(* IEC 61131-3 sources: inproshop/test8_exported/1.Function/FB/Robot(机械手)/Kuka-六轴, 4 files *)

(* ---- Str_Kuka6.st ---- *)
TYPE Str_Kuka6 :
STRUCT
	Cmd:Str_Kuka6Cmd;//控制
	Status:Str_Kuka6Status;//状态
END_STRUCT
END_TYPE

(* ---- Str_Kuka6Cmd.st ---- *)
TYPE Str_Kuka6Cmd :
STRUCT
	AppID0			:BOOL;//Main程序编号
	AppID1			:BOOL;//Main程序编号
	AppID2			:BOOL;//Main程序编号
	AppID3			:BOOL;//Main程序编号
	AppID4			:BOOL;//Main程序编号
	AppID5			:BOOL;//Main程序编号
	AppID6			:BOOL;//Main程序编号
	AppID7			:BOOL;//Main程序编号
	PGNO_VALID		:BOOL;//程序号有效
	EXT_START		:BOOL;//启动
	MOVE_ENABLE		:BOOL;//运行开通-激活运动使能
	CONF_MESS		:BOOL;//错误确认
	DRIVES_OFF		:BOOL;//驱动器关闭
	DRIVES_ON		:BOOL;//驱动装置接通
	EXT_Stop		:BOOL;//程序复位
	MachineIntial	:BOOL;//设备初始化
	MachineAutoRun	:BOOL;//设备自动中
	MachineStepRun	:BOOL;//单步信号
	SpaceBoo19		:BOOL;//预备位
	SpaceBoo20		:BOOL;//预备位
	SpaceBoo21		:BOOL;//预备位
	SpaceBoo22		:BOOL;//预备位
	SpaceBoo23		:BOOL;//预备位
	SpaceBoo24		:BOOL;//预备位
	SpaceBoo25		:BOOL;//预备位
	SpaceBoo26		:BOOL;//预备位
	SpaceBoo27		:BOOL;//预备位
	SpaceBoo28		:BOOL;//预备位
	SpaceBoo29		:BOOL;//预备位
	SpaceBoo30		:BOOL;//预备位
	SpaceBoo31		:BOOL;//预备位
	SpaceBoo32		:BOOL;//预备位
	InterFace_B		:ARRAY[33..64] OF BOOL;//交互信号
	Speed				:INT;//	运行速度(第9-10个字节)
	ProductType			:INT;//配方型号(第11-12个字节)
	StepNum				:INT;//步序号(第13-14个字节)
	InterFace_Register4	:INT;//交换数据字(第15-16个字节)
	InterFace_Register5	:INT;//交换数据字(第17-18个字节)
	InterFace_Register6	:INT;//交换数据字(第19-20个字节)
	InterFace_Register7	:INT;//交换数据字(第21-22个字节)
	InterFace_Register8	:INT;//交换数据字(第23-24个字节)
	InterFace_Register9	:INT;//交换数据字(第25-26个字节)
	InterFace_Register10	:REAL;//交换数据字(第27-30个字节)
	InterFace_Register11	:REAL;//交换数据字(第31-34个字节)
	InterFace_Register12	:REAL;//交换数据字
	InterFace_Register13	:REAL;//交换数据字
	InterFace_Register14	:REAL;//交换数据字
	InterFace_Register15	:REAL;//交换数据字
	InterFace_Register16	:REAL;//交换数据字

END_STRUCT
END_TYPE

(* ---- Str_Kuka6Status.st ---- *)
TYPE Str_Kuka6Status :
STRUCT
	AppID0			:BOOL;//返回程序编号
	AppID1			:BOOL;//返回程序编号
	AppID2			:BOOL;//返回程序编号
	AppID3			:BOOL;//返回程序编号
	AppID4			:BOOL;//返回程序编号
	AppID5			:BOOL;//返回程序编号
	AppID6			:BOOL;//返回程序编号
	AppID7			:BOOL;//返回程序编号
	ALARM_STOP:		BOOL;//	急停
	USER_SAF:		BOOL;//	安全门
	Ready:			BOOL;//	驱动器处于待机运行状态
	STOPMESS:		BOOL;//	集合故障
	PRO_ACT:		BOOL;//	程序激活
	PGNO_REQ:		BOOL;//	程序号请求
	APPL_RUN:		BOOL;//	运行中
	EXT:			BOOL;//外部自动运行
	Intialed:		BOOL;//	机械手初始化完成
	SpaceBoo18		:BOOL;//预备位
	SpaceBoo19		:BOOL;//预备位
	SpaceBoo20		:BOOL;//预备位
	SpaceBoo21		:BOOL;//预备位
	SpaceBoo22		:BOOL;//预备位
	SpaceBoo23		:BOOL;//预备位
	SpaceBoo24		:BOOL;//预备位
	SpaceBoo25		:BOOL;//预备位
	SpaceBoo26		:BOOL;//预备位
	SpaceBoo27		:BOOL;//预备位
	SpaceBoo28		:BOOL;//预备位
	SpaceBoo29		:BOOL;//预备位
	SpaceBoo30		:BOOL;//预备位
	SpaceBoo31		:BOOL;//预备位
	SpaceBoo32		:BOOL;//预备位
	InterFace_B:ARRAY[33..64] OF BOOL;//交互信号
	ErrorCode:			WORD;//	错误代码（9-10）
	ProductType			:INT;//配方型号(第11-12个字节)
	StepNum				:INT;//步序号(第13-14个字节)
	InterFace_Register19:	WORD;// 交换数据字(Holding Register19)
	InterFace_Register20:	WORD;//	交换数据字(Holding Register20)
	InterFace_Register21:	WORD;//	交换数据字(Holding Register21)
	InterFace_Register22:	WORD;//	交换数据字(Holding Register22)
	InterFace_Register23:	WORD;//	交换数据字(Holding Register23)
	InterFace_Register24:	WORD;//	交换数据字(Holding Register24)
	InterFace_Register25:	WORD;//	交换数据字(Holding Register25)
	InterFace_Register26:	WORD;//	交换数据字(Holding Register26)
	InterFace_Register27:	WORD;// 交换数据字(Holding Register27)
	InterFace_Register28:	WORD;//	交换数据字(Holding Register28)
	InterFace_Register29:	WORD;// 交换数据字(Holding Register29)
	InterFace_Register30:	WORD;//	交换数据字(Holding Register30)
	InterFace_Register31:	WORD;//	交换数据字(Holding Register31)
	InterFace_Register32:	WORD;//	交换数据字(Holding Register32)
END_STRUCT
END_TYPE

(* ---- FB_Kuka6_V1.st ---- *)
FUNCTION_BLOCK FB_Kuka6_V1
VAR_IN_OUT
	ioKuka:Str_Kuka6;
END_VAR
VAR_INPUT
	iMode:Str_Mode;//设备控制模式
	iName:WSTRING;//名称
	iSpeed:REAL;//运行速度
	iProductType:INT;//配方名称
	inputAddres:ARRAY[0..63] OF BYTE;
END_VAR
VAR_OUTPUT
	oRESET:BOOL;//安全回路复位
	outputAddres: ARRAY[0..63] OF BYTE;
	oTimeOut:BOOL;//通讯超时
END_VAR
VAR
	i:INT;//循环变量用
	TcpClient:Str_TcpClient;
	FB_TcpClient_instance:FB_TcpClient;//通讯功能块实例化
	bySendData:ARRAY[0..63]OF BYTE;
	byRevData:ARRAY[0..63]OF BYTE;
	change:INT;//切换读写状态
	TimeDelayExcute:TON;//数据发送间隔
	TimeDelayExcute_R:R_TRIG;
	TimeDelayControl:ARRAY[0..9] OF TON;//控制延时
	TimeOutDelay:TON;//超时
	EnableDelay:TON;//延时使能
END_VAR

ACT_Input();
ACT_Control();
ACT_Output();
